// TIA Portal V20 export
TYPE "typeEmHomedCheck"
// stored: Access Published, Namespace Unit1.Em4
   STRUCT
      cmCompensatorAxisZ : Bool;
      cmFeedingRollAxisB : Bool;
      cmElectrodeCutterAxisZ : Bool;
      cmPositionMovingAxisX : Bool;
   END_STRUCT;
END_TYPE
